TYPE "UDT_ZC_PREAL"
VERSION : 0.1
   STRUCT
      Valor : Real;
      ValorAnterior : Real;
      Maximo : Real;   // Límite máximo
      Minimo : Real;   // Límite mínimo
   END_STRUCT;

END_TYPE

